Staubli VAL3: SaveData.dtx

public bool bHome = true
public jointRx jJhome
public mdesc mNomSpeed
public num nPage_Traj = 1
public num nPage_editTraj = 7
public num nPage_viewTraj = 1
public pointRx pPoinTest[8]
  [0] = {x=32, y=32, fatherId=world[0]}
  [1] = {x=44, y=98, z=99, rx=55, ry=33, rz=22, fatherId=world[0]}
  [2] = {x=332, y=23, z=2, rx=23, ry=22, fatherId=world[0]}
  [3] = {y=34, rx=23, fatherId=world[0]}
  [4] = {x=12, y=22, z=90, rx=23, ry=23, rz=23, fatherId=world[0]}
  [5] = {x=11, z=44, rx=34, ry=12, rz=23, fatherId=world[0]}
  [6] = {x=2, y=22, z=4, rx=2, ry=33, rz=11, fatherId=world[0]}
  [7] = {x=23, fatherId=world[0]}
public string sTest
